# B&R Automation Studio project Lecture_07_jbl
Automation Studio 4.8.2.72

## Configuration Config1

### Task classes (Cpu.sw)
```
Cyclic#1:
  Opgave2 <- Opgave2.prg
Cyclic#6 (cycle 900000 us, tolerance 900000 us):
  Blinklys_t <- Blinklys_opg_i_timerne.prg
  Opgave1 <- Opgave1.prg
Binaries: udbdef, FWRules, TCData, sysconf, Role, User, iomap, ashwd, asfw, arconfig, ashwac
Libraries: standard, runtime, astime, asieccon
```

### Hardware
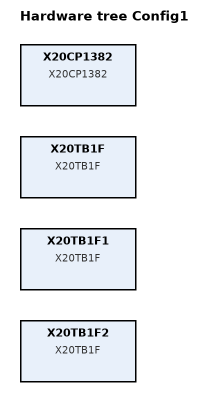
```
X20CP1382 : X20CP1382 v1.10.0.0  [X1 -> X1.SL; X2 -> X2.SL; X3 -> X3.SL]
  Module X1 (Type=X1, Virtual=true, Version=1.10.0.0)
    Connection (Connector=SS1, TargetModule=X20TB1F, TargetConnector=SS)
    Connection (Connector=SL, TargetModule=X20CP1382, TargetConnector=X1)
  Module X2 (Type=X2, Virtual=true, Version=1.10.0.0)
    Connection (Connector=SS1, TargetModule=X20TB1F1, TargetConnector=SS)
    Connection (Connector=SL, TargetModule=X20CP1382, TargetConnector=X2)
  Module X3 (Type=X3, Virtual=true, Version=1.10.0.0)
    Connection (Connector=SS1, TargetModule=X20TB1F2, TargetConnector=SS)
    Connection (Connector=SL, TargetModule=X20CP1382, TargetConnector=X3)
  Connector IF2:
    ActivateDevice = 1
  ConfigurationID = Blinklys_opgave_fra_timen_Config1
  Simulation = 1
  Cyclic6Duration = 900000
  Cyclic6Tolerance = 900000
X20TB1F : X20TB1F v1.0.0.0
X20TB1F1 : X20TB1F v1.0.0.0
X20TB1F2 : X20TB1F v1.0.0.0
```

## Logical view

### Program Logical/Blinklys_opg_i_timerne (IEC)

#### Variables.var
```iecst
VAR
	timer : TON;
	light : BOOL;
END_VAR
```

### Program Logical/Opgave1 (IEC)

#### Variables.var
```iecst
VAR
	tmp : BOOL;
	i : USINT;
	shift : BOOL;
	lights : ARRAY[0..15] OF BOOL;
END_VAR
```

#### Main.st
```iecst
PROGRAM _INIT
	(* Insert code here *)
	lights[15] := TRUE;

END_PROGRAM

PROGRAM _CYCLIC
	(* Insert code here *)

	(*
	IF (shift) THEN
		FOR i := 0 TO 15 BY 1 DO
			IF (i = 0) THEN
				lights[0] := lights[15];
				lights[15] := FALSE;
			ELSE
				lights[i] := lights[i - 1];
				lights[i - 1] := FALSE;
			END_IF;
		END_FOR;
	END_IF;
	*)

	IF shift THEN
		tmp:= lights[0];

		FOR i := 0 TO 14 BY 1 DO
			lights[i] := lights[i + 1];
		END_FOR

		lights[15] := tmp;
	END_IF

END_PROGRAM

PROGRAM _EXIT
	(* Insert code here *)

END_PROGRAM
```

### Program Logical/Opgave2 (IEC)

#### Variables.var
```iecst
VAR
	i : USINT;
	shift : BOOL;
	lights : ARRAY[0..15] OF BOOL;
	j : USINT;
	tmp : BOOL;
END_VAR
```

#### Main.st
```iecst
PROGRAM _INIT
	(* Insert code here *)
	lights[15] := TRUE;

END_PROGRAM

PROGRAM _CYCLIC
	(* Insert code here *)

	IF (shift) THEN
		FOR i := 0 TO 15 BY 1 DO
			IF (i = 0) THEN
				lights[0] := lights[15];
				lights[15] := FALSE;
			ELSE
				lights[i] := lights[i - 1];
				lights[i - 1] := FALSE;
			END_IF;
		END_FOR;
	END_IF;

			END_PROGRAM

			PROGRAM _EXIT
			(* Insert code here *)

			END_PROGRAM
```

Listed in the project but not available here: Logical/Global.typ, Logical/Global.var, Logical/Libraries
